//     Term 9 (AT2000-0250)/CC Outputs/Current setpoint value Ch.4 <-> Data Pointer/CurrentSetpointValues[3]
//     Term 9 (AT2000-0250)/CC Outputs/Current setpoint value Ch.5 <-> Data Pointer/CurrentSetpointValues[4]
//     Term 9 (AT2000-0250)/CC Outputs/Current setpoint value Ch.6 <-> Data Pointer/CurrentSetpointValues[5]
//     Term 9 (AT2000-0250)/CC Outputs/Current setpoint value Ch.7 <-> Data Pointer/CurrentSetpointValues[6]
//     Term 9 (AT2000-0250)/CC Outputs/Current setpoint value Ch.8 <-> Data Pointer/CurrentSetpointValues[7]
//     Term 9 (AT2000-0250)/CC Outputs/Current setpoint value Ch.9 <-> Data Pointer/CurrentSetpointValues[8]
//     Term 9 (AT2000-0250)/Term 10 (AT2000-5250)/FB Inputs/Value Channel 01 <-> Data Pointer/RawPositionValues[0]
//     Term 9 (AT2000-0250)/Term 10 (AT2000-5250)/FB Inputs/Value Channel 02 <-> Data Pointer/RawPositionValues[1]
//     Term 9 (AT2000-0250)/Term 10 (AT2000-5250)/FB Inputs/Value Channel 03 <-> Data Pointer/RawPositionValues[2]
//     Term 9 (AT2000-0250)/Term 10 (AT2000-5250)/FB Inputs/Value Channel 04 <-> Data Pointer/RawPositionValues[3]
//     Term 9 (AT2000-0250)/Term 10 (AT2000-5250)/FB Inputs/Value Channel 05 <-> Data Pointer/RawPositionValues[4]
//     Term 9 (AT2000-0250)/Term 10 (AT2000-5250)/FB Inputs/Value Channel 06 <-> Data Pointer/RawPositionValues[5]
//     Term 9 (AT2000-0250)/Term 10 (AT2000-5250)/FB Inputs/Value Channel 07 <-> Data Pointer/RawPositionValues[6]
//     Term 9 (AT2000-0250)/Term 10 (AT2000-5250)/FB Inputs/Value Channel 08 <-> Data Pointer/RawPositionValues[7]
//     Term 9 (AT2000-0250)/Term 10 (AT2000-5250)/FB Inputs/Value Channel 09 <-> Data Pointer/RawPositionValues[8]
//     Term 9 (AT2000-0250)/Term 10 (AT2000-5250)/FB Inputs/Value Channel 10 <-> Data Pointer/RawPositionValues[9]
//     Term 9 (AT2000-0250)/Term 10 (AT2000-5250)/FB Inputs/Value Channel 11 <-> Data Pointer/RawPositionValues[10]
//     Term 9 (AT2000-0250)/Term 10 (AT2000-5250)/FB Inputs/Value Channel 12 <-> Data Pointer/RawPositionValues[11]
//     Term 9 (AT2000-0250)/Term 10 (AT2000-5250)/FB Inputs/Value Channel 13 <-> Data Pointer/RawPositionValues[12]
//     Term 9 (AT2000-0250)/Term 10 (AT2000-5250)/FB Inputs/Value Channel 14 <-> Data Pointer/RawPositionValues[13]
//     Term 9 (AT2000-0250)/Term 10 (AT2000-5250)/FB Inputs/Value Channel 15 <-> Data Pointer/RawPositionValues[14]
//     Term 9 (AT2000-0250)/Term 10 (AT2000-5250)/FB Inputs/Value Channel 16 <-> Data Pointer/RawPositionValues[15]
//     Term 9 (AT2000-0250)/Term 10 (AT2000-5250)/FB Inputs/Value Channel 17 <-> Data Pointer/RawPositionValues[16]
//     Term 9 (AT2000-0250)/Term 10 (AT2000-5250)/FB Inputs/Value Channel 18 <-> Data Pointer/RawPositionValues[17]
//     Term 9 (AT2000-0250)/Term 10 (AT2000-5250)/FB Inputs/Value Channel 19 <-> Data Pointer/RawPositionValues[18]
//     Term 9 (AT2000-0250)/Term 10 (AT2000-5250)/FB Inputs/Value Channel 20 <-> Data Pointer/RawPositionValues[19]
//     Term 9 (AT2000-0250)/Term 10 (AT2000-5250)/FB Inputs/Value Channel 21 <-> Data Pointer/RawPositionValues[20]
//     Term 9 (AT2000-0250)/Term 10 (AT2000-5250)/FB Inputs/Value Channel 22 <-> Data Pointer/RawPositionValues[21]
//     Term 9 (AT2000-0250)/Term 10 (AT2000-5250)/FB Inputs/Value Channel 23 <-> Data Pointer/RawPositionValues[22]
//     Term 9 (AT2000-0250)/Term 10 (AT2000-5250)/FB Inputs/Value Channel 24 <-> Data Pointer/RawPositionValues[23]
//     Term 9 (AT2000-0250)/Term 10 (AT2000-5250)/FB Inputs/Value Channel 25 <-> Data Pointer/RawPositionValues[24]
//     Term 9 (AT2000-0250)/Term 10 (AT2000-5250)/FB Inputs/Value Channel 26 <-> Data Pointer/RawPositionValues[25]
//     Term 9 (AT2000-0250)/Term 10 (AT2000-5250)/FB Inputs/Value Channel 27 <-> Data Pointer/RawPositionValues[26]
//     Term 9 (AT2000-0250)/Term 10 (AT2000-5250)/FB Inputs/Value Channel 28 <-> Data Pointer/RawPositionValues[27]
//     Term 9 (AT2000-0250)/Term 10 (AT2000-5250)/FB Inputs/Value Channel 29 <-> Data Pointer/RawPositionValues[28]
//     Term 9 (AT2000-0250)/Term 10 (AT2000-5250)/FB Inputs/Value Channel 30 <-> Data Pointer/RawPositionValues[29]
//     Term 9 (AT2000-0250)/Term 10 (AT2000-5250)/FB Inputs/Value Channel 31 <-> Data Pointer/RawPositionValues[30]
//     Term 9 (AT2000-0250)/Term 10 (AT2000-5250)/FB Inputs/Value Channel 32 <-> Data Pointer/RawPositionValues[31]
//   (this object) <-> TcCOM Objects/XtsProcessingUnit 1/Part 1/Module 6
//     Term 11 (AT2000-0250)/CC Inputs/Current actual value Ch.1 <-> Data Pointer/CurrentActualValues[0]
//     Term 11 (AT2000-0250)/CC Inputs/Current actual value Ch.10 <-> Data Pointer/CurrentActualValues[9]
//     Term 11 (AT2000-0250)/CC Inputs/Current actual value Ch.11 <-> Data Pointer/CurrentActualValues[10]
//     Term 11 (AT2000-0250)/CC Inputs/Current actual value Ch.12 <-> Data Pointer/CurrentActualValues[11]
//     Term 11 (AT2000-0250)/CC Inputs/Current actual value Ch.13 <-> Data Pointer/CurrentActualValues[12]
//     Term 11 (AT2000-0250)/CC Inputs/Current actual value Ch.14 <-> Data Pointer/CurrentActualValues[13]
//     Term 11 (AT2000-0250)/CC Inputs/Current actual value Ch.15 <-> Data Pointer/CurrentActualValues[14]
//     Term 11 (AT2000-0250)/CC Inputs/Current actual value Ch.2 <-> Data Pointer/CurrentActualValues[1]
//     Term 11 (AT2000-0250)/CC Inputs/Current actual value Ch.3 <-> Data Pointer/CurrentActualValues[2]
//     Term 11 (AT2000-0250)/CC Inputs/Current actual value Ch.4 <-> Data Pointer/CurrentActualValues[3]
//     Term 11 (AT2000-0250)/CC Inputs/Current actual value Ch.5 <-> Data Pointer/CurrentActualValues[4]
//     Term 11 (AT2000-0250)/CC Inputs/Current actual value Ch.6 <-> Data Pointer/CurrentActualValues[5]
//     Term 11 (AT2000-0250)/CC Inputs/Current actual value Ch.7 <-> Data Pointer/CurrentActualValues[6]
//     Term 11 (AT2000-0250)/CC Inputs/Current actual value Ch.8 <-> Data Pointer/CurrentActualValues[7]
//     Term 11 (AT2000-0250)/CC Inputs/Current actual value Ch.9 <-> Data Pointer/CurrentActualValues[8]
//     Term 11 (AT2000-0250)/CC Inputs/Status <-> Data Pointer/Status
//     Term 11 (AT2000-0250)/CC Outputs/Control <-> Data Pointer/Control
//     Term 11 (AT2000-0250)/CC Outputs/Current setpoint value Ch.1 <-> Data Pointer/CurrentSetpointValues[0]
//     Term 11 (AT2000-0250)/CC Outputs/Current setpoint value Ch.10 <-> Data Pointer/CurrentSetpointValues[9]
//     Term 11 (AT2000-0250)/CC Outputs/Current setpoint value Ch.11 <-> Data Pointer/CurrentSetpointValues[10]
//     Term 11 (AT2000-0250)/CC Outputs/Current setpoint value Ch.12 <-> Data Pointer/CurrentSetpointValues[11]
//     Term 11 (AT2000-0250)/CC Outputs/Current setpoint value Ch.13 <-> Data Pointer/CurrentSetpointValues[12]
//     Term 11 (AT2000-0250)/CC Outputs/Current setpoint value Ch.14 <-> Data Pointer/CurrentSetpointValues[13]
//     Term 11 (AT2000-0250)/CC Outputs/Current setpoint value Ch.15 <-> Data Pointer/CurrentSetpointValues[14]
//     Term 11 (AT2000-0250)/CC Outputs/Current setpoint value Ch.2 <-> Data Pointer/CurrentSetpointValues[1]
//     Term 11 (AT2000-0250)/CC Outputs/Current setpoint value Ch.3 <-> Data Pointer/CurrentSetpointValues[2]
//     Term 11 (AT2000-0250)/CC Outputs/Current setpoint value Ch.4 <-> Data Pointer/CurrentSetpointValues[3]
//     Term 11 (AT2000-0250)/CC Outputs/Current setpoint value Ch.5 <-> Data Pointer/CurrentSetpointValues[4]
//     Term 11 (AT2000-0250)/CC Outputs/Current setpoint value Ch.6 <-> Data Pointer/CurrentSetpointValues[5]
//     Term 11 (AT2000-0250)/CC Outputs/Current setpoint value Ch.7 <-> Data Pointer/CurrentSetpointValues[6]
//     Term 11 (AT2000-0250)/CC Outputs/Current setpoint value Ch.8 <-> Data Pointer/CurrentSetpointValues[7]
//     Term 11 (AT2000-0250)/CC Outputs/Current setpoint value Ch.9 <-> Data Pointer/CurrentSetpointValues[8]
//     Term 11 (AT2000-0250)/Term 12 (AT2000-5250)/FB Inputs/Value Channel 01 <-> Data Pointer/RawPositionValues[0]
//     Term 11 (AT2000-0250)/Term 12 (AT2000-5250)/FB Inputs/Value Channel 02 <-> Data Pointer/RawPositionValues[1]
//     Term 11 (AT2000-0250)/Term 12 (AT2000-5250)/FB Inputs/Value Channel 03 <-> Data Pointer/RawPositionValues[2]
//     Term 11 (AT2000-0250)/Term 12 (AT2000-5250)/FB Inputs/Value Channel 04 <-> Data Pointer/RawPositionValues[3]
//     Term 11 (AT2000-0250)/Term 12 (AT2000-5250)/FB Inputs/Value Channel 05 <-> Data Pointer/RawPositionValues[4]
//     Term 11 (AT2000-0250)/Term 12 (AT2000-5250)/FB Inputs/Value Channel 06 <-> Data Pointer/RawPositionValues[5]
//     Term 11 (AT2000-0250)/Term 12 (AT2000-5250)/FB Inputs/Value Channel 07 <-> Data Pointer/RawPositionValues[6]
//     Term 11 (AT2000-0250)/Term 12 (AT2000-5250)/FB Inputs/Value Channel 08 <-> Data Pointer/RawPositionValues[7]
//     Term 11 (AT2000-0250)/Term 12 (AT2000-5250)/FB Inputs/Value Channel 09 <-> Data Pointer/RawPositionValues[8]
//     Term 11 (AT2000-0250)/Term 12 (AT2000-5250)/FB Inputs/Value Channel 10 <-> Data Pointer/RawPositionValues[9]
//     Term 11 (AT2000-0250)/Term 12 (AT2000-5250)/FB Inputs/Value Channel 11 <-> Data Pointer/RawPositionValues[10]
//     Term 11 (AT2000-0250)/Term 12 (AT2000-5250)/FB Inputs/Value Channel 12 <-> Data Pointer/RawPositionValues[11]
//     Term 11 (AT2000-0250)/Term 12 (AT2000-5250)/FB Inputs/Value Channel 13 <-> Data Pointer/RawPositionValues[12]
//     Term 11 (AT2000-0250)/Term 12 (AT2000-5250)/FB Inputs/Value Channel 14 <-> Data Pointer/RawPositionValues[13]
//     Term 11 (AT2000-0250)/Term 12 (AT2000-5250)/FB Inputs/Value Channel 15 <-> Data Pointer/RawPositionValues[14]
//     Term 11 (AT2000-0250)/Term 12 (AT2000-5250)/FB Inputs/Value Channel 16 <-> Data Pointer/RawPositionValues[15]
//     Term 11 (AT2000-0250)/Term 12 (AT2000-5250)/FB Inputs/Value Channel 17 <-> Data Pointer/RawPositionValues[16]
//     Term 11 (AT2000-0250)/Term 12 (AT2000-5250)/FB Inputs/Value Channel 18 <-> Data Pointer/RawPositionValues[17]
//     Term 11 (AT2000-0250)/Term 12 (AT2000-5250)/FB Inputs/Value Channel 19 <-> Data Pointer/RawPositionValues[18]
//     Term 11 (AT2000-0250)/Term 12 (AT2000-5250)/FB Inputs/Value Channel 20 <-> Data Pointer/RawPositionValues[19]
//     Term 11 (AT2000-0250)/Term 12 (AT2000-5250)/FB Inputs/Value Channel 21 <-> Data Pointer/RawPositionValues[20]
//     Term 11 (AT2000-0250)/Term 12 (AT2000-5250)/FB Inputs/Value Channel 22 <-> Data Pointer/RawPositionValues[21]
//     Term 11 (AT2000-0250)/Term 12 (AT2000-5250)/FB Inputs/Value Channel 23 <-> Data Pointer/RawPositionValues[22]
//     Term 11 (AT2000-0250)/Term 12 (AT2000-5250)/FB Inputs/Value Channel 24 <-> Data Pointer/RawPositionValues[23]
//     Term 11 (AT2000-0250)/Term 12 (AT2000-5250)/FB Inputs/Value Channel 25 <-> Data Pointer/RawPositionValues[24]
//     Term 11 (AT2000-0250)/Term 12 (AT2000-5250)/FB Inputs/Value Channel 26 <-> Data Pointer/RawPositionValues[25]
//     Term 11 (AT2000-0250)/Term 12 (AT2000-5250)/FB Inputs/Value Channel 27 <-> Data Pointer/RawPositionValues[26]
//     Term 11 (AT2000-0250)/Term 12 (AT2000-5250)/FB Inputs/Value Channel 28 <-> Data Pointer/RawPositionValues[27]
//     Term 11 (AT2000-0250)/Term 12 (AT2000-5250)/FB Inputs/Value Channel 29 <-> Data Pointer/RawPositionValues[28]
//     Term 11 (AT2000-0250)/Term 12 (AT2000-5250)/FB Inputs/Value Channel 30 <-> Data Pointer/RawPositionValues[29]
//     Term 11 (AT2000-0250)/Term 12 (AT2000-5250)/FB Inputs/Value Channel 31 <-> Data Pointer/RawPositionValues[30]
//     Term 11 (AT2000-0250)/Term 12 (AT2000-5250)/FB Inputs/Value Channel 32 <-> Data Pointer/RawPositionValues[31]
//   (this object) <-> TcCOM Objects/XtsProcessingUnit 1/Part 1/Module 7
//     Term 13 (AT2050-0500)/CC Inputs/Current actual value Ch.1 <-> Data Pointer/CurrentActualValues[0]
//     Term 13 (AT2050-0500)/CC Inputs/Current actual value Ch.10 <-> Data Pointer/CurrentActualValues[9]
//     Term 13 (AT2050-0500)/CC Inputs/Current actual value Ch.11 <-> Data Pointer/CurrentActualValues[10]
//     Term 13 (AT2050-0500)/CC Inputs/Current actual value Ch.12 <-> Data Pointer/CurrentActualValues[11]
//     Term 13 (AT2050-0500)/CC Inputs/Current actual value Ch.13 <-> Data Pointer/CurrentActualValues[12]
//     Term 13 (AT2050-0500)/CC Inputs/Current actual value Ch.14 <-> Data Pointer/CurrentActualValues[13]
//     Term 13 (AT2050-0500)/CC Inputs/Current actual value Ch.15 <-> Data Pointer/CurrentActualValues[14]
//     Term 13 (AT2050-0500)/CC Inputs/Current actual value Ch.2 <-> Data Pointer/CurrentActualValues[1]
//     Term 13 (AT2050-0500)/CC Inputs/Current actual value Ch.3 <-> Data Pointer/CurrentActualValues[2]
//     Term 13 (AT2050-0500)/CC Inputs/Current actual value Ch.4 <-> Data Pointer/CurrentActualValues[3]
//     Term 13 (AT2050-0500)/CC Inputs/Current actual value Ch.5 <-> Data Pointer/CurrentActualValues[4]
//     Term 13 (AT2050-0500)/CC Inputs/Current actual value Ch.6 <-> Data Pointer/CurrentActualValues[5]
//     Term 13 (AT2050-0500)/CC Inputs/Current actual value Ch.7 <-> Data Pointer/CurrentActualValues[6]
//     Term 13 (AT2050-0500)/CC Inputs/Current actual value Ch.8 <-> Data Pointer/CurrentActualValues[7]
//     Term 13 (AT2050-0500)/CC Inputs/Current actual value Ch.9 <-> Data Pointer/CurrentActualValues[8]
//     Term 13 (AT2050-0500)/CC Inputs/Status <-> Data Pointer/Status
//     Term 13 (AT2050-0500)/CC Outputs/Control <-> Data Pointer/Control
//     Term 13 (AT2050-0500)/CC Outputs/Current setpoint value Ch.1 <-> Data Pointer/CurrentSetpointValues[0]
//     Term 13 (AT2050-0500)/CC Outputs/Current setpoint value Ch.10 <-> Data Pointer/CurrentSetpointValues[9]
//     Term 13 (AT2050-0500)/CC Outputs/Current setpoint value Ch.11 <-> Data Pointer/CurrentSetpointValues[10]
//     Term 13 (AT2050-0500)/CC Outputs/Current setpoint value Ch.12 <-> Data Pointer/CurrentSetpointValues[11]
//     Term 13 (AT2050-0500)/CC Outputs/Current setpoint value Ch.13 <-> Data Pointer/CurrentSetpointValues[12]
//     Term 13 (AT2050-0500)/CC Outputs/Current setpoint value Ch.14 <-> Data Pointer/CurrentSetpointValues[13]
//     Term 13 (AT2050-0500)/CC Outputs/Current setpoint value Ch.15 <-> Data Pointer/CurrentSetpointValues[14]
//     Term 13 (AT2050-0500)/CC Outputs/Current setpoint value Ch.2 <-> Data Pointer/CurrentSetpointValues[1]
//     Term 13 (AT2050-0500)/CC Outputs/Current setpoint value Ch.3 <-> Data Pointer/CurrentSetpointValues[2]
//     Term 13 (AT2050-0500)/CC Outputs/Current setpoint value Ch.4 <-> Data Pointer/CurrentSetpointValues[3]
//     Term 13 (AT2050-0500)/CC Outputs/Current setpoint value Ch.5 <-> Data Pointer/CurrentSetpointValues[4]
//     Term 13 (AT2050-0500)/CC Outputs/Current setpoint value Ch.6 <-> Data Pointer/CurrentSetpointValues[5]
//     Term 13 (AT2050-0500)/CC Outputs/Current setpoint value Ch.7 <-> Data Pointer/CurrentSetpointValues[6]
//     Term 13 (AT2050-0500)/CC Outputs/Current setpoint value Ch.8 <-> Data Pointer/CurrentSetpointValues[7]
//     Term 13 (AT2050-0500)/CC Outputs/Current setpoint value Ch.9 <-> Data Pointer/CurrentSetpointValues[8]
//     Term 13 (AT2050-0500)/Term 14 (AT2050-5500)/FB Inputs/Value Channel 01 <-> Data Pointer/RawPositionValues[0]
//     Term 13 (AT2050-0500)/Term 14 (AT2050-5500)/FB Inputs/Value Channel 02 <-> Data Pointer/RawPositionValues[1]
//     Term 13 (AT2050-0500)/Term 14 (AT2050-5500)/FB Inputs/Value Channel 03 <-> Data Pointer/RawPositionValues[2]
//     Term 13 (AT2050-0500)/Term 14 (AT2050-5500)/FB Inputs/Value Channel 04 <-> Data Pointer/RawPositionValues[3]
//     Term 13 (AT2050-0500)/Term 14 (AT2050-5500)/FB Inputs/Value Channel 05 <-> Data Pointer/RawPositionValues[4]
//     Term 13 (AT2050-0500)/Term 14 (AT2050-5500)/FB Inputs/Value Channel 06 <-> Data Pointer/RawPositionValues[5]
//     Term 13 (AT2050-0500)/Term 14 (AT2050-5500)/FB Inputs/Value Channel 07 <-> Data Pointer/RawPositionValues[6]
//     Term 13 (AT2050-0500)/Term 14 (AT2050-5500)/FB Inputs/Value Channel 08 <-> Data Pointer/RawPositionValues[7]
//     Term 13 (AT2050-0500)/Term 14 (AT2050-5500)/FB Inputs/Value Channel 09 <-> Data Pointer/RawPositionValues[8]
//     Term 13 (AT2050-0500)/Term 14 (AT2050-5500)/FB Inputs/Value Channel 10 <-> Data Pointer/RawPositionValues[9]
//     Term 13 (AT2050-0500)/Term 14 (AT2050-5500)/FB Inputs/Value Channel 11 <-> Data Pointer/RawPositionValues[10]
//     Term 13 (AT2050-0500)/Term 14 (AT2050-5500)/FB Inputs/Value Channel 12 <-> Data Pointer/RawPositionValues[11]
//     Term 13 (AT2050-0500)/Term 14 (AT2050-5500)/FB Inputs/Value Channel 13 <-> Data Pointer/RawPositionValues[12]
//     Term 13 (AT2050-0500)/Term 14 (AT2050-5500)/FB Inputs/Value Channel 14 <-> Data Pointer/RawPositionValues[13]
//     Term 13 (AT2050-0500)/Term 14 (AT2050-5500)/FB Inputs/Value Channel 15 <-> Data Pointer/RawPositionValues[14]
//     Term 13 (AT2050-0500)/Term 14 (AT2050-5500)/FB Inputs/Value Channel 16 <-> Data Pointer/RawPositionValues[15]
//     Term 13 (AT2050-0500)/Term 14 (AT2050-5500)/FB Inputs/Value Channel 17 <-> Data Pointer/RawPositionValues[16]
//     Term 13 (AT2050-0500)/Term 14 (AT2050-5500)/FB Inputs/Value Channel 18 <-> Data Pointer/RawPositionValues[17]
//     Term 13 (AT2050-0500)/Term 14 (AT2050-5500)/FB Inputs/Value Channel 19 <-> Data Pointer/RawPositionValues[18]
//     Term 13 (AT2050-0500)/Term 14 (AT2050-5500)/FB Inputs/Value Channel 20 <-> Data Pointer/RawPositionValues[19]
//     Term 13 (AT2050-0500)/Term 14 (AT2050-5500)/FB Inputs/Value Channel 21 <-> Data Pointer/RawPositionValues[20]
//     Term 13 (AT2050-0500)/Term 14 (AT2050-5500)/FB Inputs/Value Channel 22 <-> Data Pointer/RawPositionValues[21]
//     Term 13 (AT2050-0500)/Term 14 (AT2050-5500)/FB Inputs/Value Channel 23 <-> Data Pointer/RawPositionValues[22]
//     Term 13 (AT2050-0500)/Term 14 (AT2050-5500)/FB Inputs/Value Channel 24 <-> Data Pointer/RawPositionValues[23]
//     Term 13 (AT2050-0500)/Term 14 (AT2050-5500)/FB Inputs/Value Channel 25 <-> Data Pointer/RawPositionValues[24]
//     Term 13 (AT2050-0500)/Term 14 (AT2050-5500)/FB Inputs/Value Channel 26 <-> Data Pointer/RawPositionValues[25]
//     Term 13 (AT2050-0500)/Term 14 (AT2050-5500)/FB Inputs/Value Channel 27 <-> Data Pointer/RawPositionValues[26]
//     Term 13 (AT2050-0500)/Term 14 (AT2050-5500)/FB Inputs/Value Channel 28 <-> Data Pointer/RawPositionValues[27]
//     Term 13 (AT2050-0500)/Term 14 (AT2050-5500)/FB Inputs/Value Channel 29 <-> Data Pointer/RawPositionValues[28]
//     Term 13 (AT2050-0500)/Term 14 (AT2050-5500)/FB Inputs/Value Channel 30 <-> Data Pointer/RawPositionValues[29]
//     Term 13 (AT2050-0500)/Term 14 (AT2050-5500)/FB Inputs/Value Channel 31 <-> Data Pointer/RawPositionValues[30]
//     Term 13 (AT2050-0500)/Term 14 (AT2050-5500)/FB Inputs/Value Channel 32 <-> Data Pointer/RawPositionValues[31]
//   (this object) <-> TcCOM Objects/XtsProcessingUnit 1/Part 1/Module 8
//     Term 15 (AT2050-0501)/CC Inputs/Current actual value Ch.1 <-> Data Pointer/CurrentActualValues[0]
//     Term 15 (AT2050-0501)/CC Inputs/Current actual value Ch.10 <-> Data Pointer/CurrentActualValues[9]
//     Term 15 (AT2050-0501)/CC Inputs/Current actual value Ch.11 <-> Data Pointer/CurrentActualValues[10]
//     Term 15 (AT2050-0501)/CC Inputs/Current actual value Ch.12 <-> Data Pointer/CurrentActualValues[11]
//     Term 15 (AT2050-0501)/CC Inputs/Current actual value Ch.13 <-> Data Pointer/CurrentActualValues[12]
//     Term 15 (AT2050-0501)/CC Inputs/Current actual value Ch.14 <-> Data Pointer/CurrentActualValues[13]
//     Term 15 (AT2050-0501)/CC Inputs/Current actual value Ch.15 <-> Data Pointer/CurrentActualValues[14]
//     Term 15 (AT2050-0501)/CC Inputs/Current actual value Ch.2 <-> Data Pointer/CurrentActualValues[1]
//     Term 15 (AT2050-0501)/CC Inputs/Current actual value Ch.3 <-> Data Pointer/CurrentActualValues[2]
//     Term 15 (AT2050-0501)/CC Inputs/Current actual value Ch.4 <-> Data Pointer/CurrentActualValues[3]
//     Term 15 (AT2050-0501)/CC Inputs/Current actual value Ch.5 <-> Data Pointer/CurrentActualValues[4]
//     Term 15 (AT2050-0501)/CC Inputs/Current actual value Ch.6 <-> Data Pointer/CurrentActualValues[5]
//     Term 15 (AT2050-0501)/CC Inputs/Current actual value Ch.7 <-> Data Pointer/CurrentActualValues[6]
//     Term 15 (AT2050-0501)/CC Inputs/Current actual value Ch.8 <-> Data Pointer/CurrentActualValues[7]
//     Term 15 (AT2050-0501)/CC Inputs/Current actual value Ch.9 <-> Data Pointer/CurrentActualValues[8]
//     Term 15 (AT2050-0501)/CC Inputs/Status <-> Data Pointer/Status
//     Term 15 (AT2050-0501)/CC Outputs/Control <-> Data Pointer/Control
//     Term 15 (AT2050-0501)/CC Outputs/Current setpoint value Ch.1 <-> Data Pointer/CurrentSetpointValues[0]
//     Term 15 (AT2050-0501)/CC Outputs/Current setpoint value Ch.10 <-> Data Pointer/CurrentSetpointValues[9]
//     Term 15 (AT2050-0501)/CC Outputs/Current setpoint value Ch.11 <-> Data Pointer/CurrentSetpointValues[10]
//     Term 15 (AT2050-0501)/CC Outputs/Current setpoint value Ch.12 <-> Data Pointer/CurrentSetpointValues[11]
//     Term 15 (AT2050-0501)/CC Outputs/Current setpoint value Ch.13 <-> Data Pointer/CurrentSetpointValues[12]
//     Term 15 (AT2050-0501)/CC Outputs/Current setpoint value Ch.14 <-> Data Pointer/CurrentSetpointValues[13]
//     Term 15 (AT2050-0501)/CC Outputs/Current setpoint value Ch.15 <-> Data Pointer/CurrentSetpointValues[14]
//     Term 15 (AT2050-0501)/CC Outputs/Current setpoint value Ch.2 <-> Data Pointer/CurrentSetpointValues[1]
//     Term 15 (AT2050-0501)/CC Outputs/Current setpoint value Ch.3 <-> Data Pointer/CurrentSetpointValues[2]
//     Term 15 (AT2050-0501)/CC Outputs/Current setpoint value Ch.4 <-> Data Pointer/CurrentSetpointValues[3]
//     Term 15 (AT2050-0501)/CC Outputs/Current setpoint value Ch.5 <-> Data Pointer/CurrentSetpointValues[4]
//     Term 15 (AT2050-0501)/CC Outputs/Current setpoint value Ch.6 <-> Data Pointer/CurrentSetpointValues[5]
//     Term 15 (AT2050-0501)/CC Outputs/Current setpoint value Ch.7 <-> Data Pointer/CurrentSetpointValues[6]
//     Term 15 (AT2050-0501)/CC Outputs/Current setpoint value Ch.8 <-> Data Pointer/CurrentSetpointValues[7]
//     Term 15 (AT2050-0501)/CC Outputs/Current setpoint value Ch.9 <-> Data Pointer/CurrentSetpointValues[8]
//     Term 15 (AT2050-0501)/Term 16 (AT2050-5501)/FB Inputs/Value Channel 01 <-> Data Pointer/RawPositionValues[0]
//     Term 15 (AT2050-0501)/Term 16 (AT2050-5501)/FB Inputs/Value Channel 02 <-> Data Pointer/RawPositionValues[1]
//     Term 15 (AT2050-0501)/Term 16 (AT2050-5501)/FB Inputs/Value Channel 03 <-> Data Pointer/RawPositionValues[2]
//     Term 15 (AT2050-0501)/Term 16 (AT2050-5501)/FB Inputs/Value Channel 04 <-> Data Pointer/RawPositionValues[3]
//     Term 15 (AT2050-0501)/Term 16 (AT2050-5501)/FB Inputs/Value Channel 05 <-> Data Pointer/RawPositionValues[4]
//     Term 15 (AT2050-0501)/Term 16 (AT2050-5501)/FB Inputs/Value Channel 06 <-> Data Pointer/RawPositionValues[5]
//     Term 15 (AT2050-0501)/Term 16 (AT2050-5501)/FB Inputs/Value Channel 07 <-> Data Pointer/RawPositionValues[6]
//     Term 15 (AT2050-0501)/Term 16 (AT2050-5501)/FB Inputs/Value Channel 08 <-> Data Pointer/RawPositionValues[7]
//     Term 15 (AT2050-0501)/Term 16 (AT2050-5501)/FB Inputs/Value Channel 09 <-> Data Pointer/RawPositionValues[8]
//     Term 15 (AT2050-0501)/Term 16 (AT2050-5501)/FB Inputs/Value Channel 10 <-> Data Pointer/RawPositionValues[9]
//     Term 15 (AT2050-0501)/Term 16 (AT2050-5501)/FB Inputs/Value Channel 11 <-> Data Pointer/RawPositionValues[10]
//     Term 15 (AT2050-0501)/Term 16 (AT2050-5501)/FB Inputs/Value Channel 12 <-> Data Pointer/RawPositionValues[11]
//     Term 15 (AT2050-0501)/Term 16 (AT2050-5501)/FB Inputs/Value Channel 13 <-> Data Pointer/RawPositionValues[12]
//     Term 15 (AT2050-0501)/Term 16 (AT2050-5501)/FB Inputs/Value Channel 14 <-> Data Pointer/RawPositionValues[13]
//     Term 15 (AT2050-0501)/Term 16 (AT2050-5501)/FB Inputs/Value Channel 15 <-> Data Pointer/RawPositionValues[14]
//     Term 15 (AT2050-0501)/Term 16 (AT2050-5501)/FB Inputs/Value Channel 16 <-> Data Pointer/RawPositionValues[15]
//     Term 15 (AT2050-0501)/Term 16 (AT2050-5501)/FB Inputs/Value Channel 17 <-> Data Pointer/RawPositionValues[16]
//     Term 15 (AT2050-0501)/Term 16 (AT2050-5501)/FB Inputs/Value Channel 18 <-> Data Pointer/RawPositionValues[17]
//     Term 15 (AT2050-0501)/Term 16 (AT2050-5501)/FB Inputs/Value Channel 19 <-> Data Pointer/RawPositionValues[18]
//     Term 15 (AT2050-0501)/Term 16 (AT2050-5501)/FB Inputs/Value Channel 20 <-> Data Pointer/RawPositionValues[19]
//     Term 15 (AT2050-0501)/Term 16 (AT2050-5501)/FB Inputs/Value Channel 21 <-> Data Pointer/RawPositionValues[20]
//     Term 15 (AT2050-0501)/Term 16 (AT2050-5501)/FB Inputs/Value Channel 22 <-> Data Pointer/RawPositionValues[21]
//     Term 15 (AT2050-0501)/Term 16 (AT2050-5501)/FB Inputs/Value Channel 23 <-> Data Pointer/RawPositionValues[22]
//     Term 15 (AT2050-0501)/Term 16 (AT2050-5501)/FB Inputs/Value Channel 24 <-> Data Pointer/RawPositionValues[23]
//     Term 15 (AT2050-0501)/Term 16 (AT2050-5501)/FB Inputs/Value Channel 25 <-> Data Pointer/RawPositionValues[24]
//     Term 15 (AT2050-0501)/Term 16 (AT2050-5501)/FB Inputs/Value Channel 26 <-> Data Pointer/RawPositionValues[25]
//     Term 15 (AT2050-0501)/Term 16 (AT2050-5501)/FB Inputs/Value Channel 27 <-> Data Pointer/RawPositionValues[26]
//     Term 15 (AT2050-0501)/Term 16 (AT2050-5501)/FB Inputs/Value Channel 28 <-> Data Pointer/RawPositionValues[27]
//     Term 15 (AT2050-0501)/Term 16 (AT2050-5501)/FB Inputs/Value Channel 29 <-> Data Pointer/RawPositionValues[28]
//     Term 15 (AT2050-0501)/Term 16 (AT2050-5501)/FB Inputs/Value Channel 30 <-> Data Pointer/RawPositionValues[29]
//     Term 15 (AT2050-0501)/Term 16 (AT2050-5501)/FB Inputs/Value Channel 31 <-> Data Pointer/RawPositionValues[30]
//     Term 15 (AT2050-0501)/Term 16 (AT2050-5501)/FB Inputs/Value Channel 32 <-> Data Pointer/RawPositionValues[31]

// ---- GVLs/Param.TcGVL
{attribute 'qualified_only'}
VAR_GLOBAL CONSTANT
	// The following should be set to a value **equal to or greater than** the number of objects needed
	MAX_MOVERS   			: USINT := 100;	// Movers
	MAX_POSITIONTRIGGERS	: USINT := 100;	// Position triggers
	MAX_STATIONS			: USINT := 100;	// Stations
	MAX_ZONES				: USINT := 100;	// Zones
	
	// The following should be set to a value **equal to or greater than** the number of objectives needed
	// it's also possible to declare additional stations, zones and position triggers in MAIN
	NUM_MOVERLISTS			: USINT := 10;	// Mover Lists
	NUM_POSITIONTRIGGERS	: USINT := 10;	// Position Triggers
	NUM_STATIONS			: USINT := 10;	// Stations
	NUM_ZONES				: USINT := 10;	// Zones
	
	NUM_TRACKS				: USINT	:= 1;	// Tracks (Typically 1)
	DEFAULT_TRACK			: USINT := 1;	// Default track for movers, stations, zones and position triggers

	PART_ARRAY_SIZE			: UDINT := 100;
	AUTO_POPULATE_STATIONS  : BOOL := TRUE; // use the Station[x] array to label stations on the visualization. Turn off if manually entering stations in the configurator.
	
	// statistics weighted average
	ALPHA_EMA				: LREAL := 0.1;
END_VAR

// ---- POUs/MAIN.TcPOU

      PROGRAM MAIN
VAR	
	// declare XTS with <number of movers>
	XTS				: FB_XTS<6>;
	// Machine
	State			: MachineState_enum;

	// ========= Example Application Variables =========

    nextStation 			: USINT := 4;
                    	
	StationTimer 			: ARRAY[0..Param.NUM_STATIONS] OF TON; // timer blocks, for station dwells
	RecoveryComplete		: BOOL;
	
	Trig0MoverIndex			: UDINT;
	Trig0MoverPosLag		: LREAL;
END_VAR


        
(* ======================================================================================

--- XTS Starter Project ---

This MAIN (PRG) is intended to serve as an example, which can be modified to suit your specific application.

No programming changes should be necessary inside the provided XTS objects / function block definitions.
They are intended to be simply instantiated and controlled via the provided methods and properties.
However the objects are provided as open-source for modification and extension as needed.

Documentation for these objects can be found online at:
https://beckhoff-usa-community.github.io/XTS_Base/

Bug reports, new feature requests, and general feedback is always welcome on our Github page.
For any other questions, please reach out to your local Application Engineer.

Version 2.1.0 of XTS_Base has been tested with:

- TwinCAT XAE v4026.20.1
- TF5850 XTS v4.4.5
- TF5410 Advanced Motion v3.4.19

- XTS Application Group | Beckhoff USA

====================================================================================== *)

(*
All sample code provided by Beckhoff Automation LLC are for illustrative purposes only
and are provided “as is” and without any warranties, express or implied. Actual
implementations in applications will vary significantly. Beckhoff Automation LLC shall
have no liability for, and does not waive any rights in relation to, any code samples that it
provides or the use of such code samples for any purpose.
*)

// main state machine
CASE State OF 

	// off (idle) state, waiting for enable command
	MS_OFF:
		// wait for enable command
		IF MainCommands.Enable AND XTS.System.EnvironmentIsReady THEN
			// initialize stations, positions and triggers
			Initializing();
			// enable the XTS
			XTS.Enable				:= TRUE;
			State					:= MS_RESTARTING;
		END_IF
		
	MS_RESTARTING:
		// restart the system by enabling the XTS and waiting for it to complete
		IF NOT MainCommands.Enable THEN
			// disable triggered, pass to xts and stop the movers
			XTS.Enable				:= FALSE;
			State					:= MS_STOPPED;
		ELSIF XTS.State = XTS_ENABLED THEN
			// enable complete move to enabled
			State		:= MS_ENABLED;
		END_IF


	MS_ENABLED:
		// XTS is enabled, wait for start command
		IF NOT MainCommands.Enable THEN
			XTS.Enable				:= FALSE;
			State					:= MS_STOPPED;
		ELSIF MainCommands.Start THEN
			// reset the recovery complete flag
			RecoveryComplete		:= FALSE;
			// move to next state
			State					:= MS_ONESHOT_RECOVER;
		END_IF
		
	MS_ONESHOT_RECOVER:
		// one time commands before starting typical process motions
		RecoverOneshot();
		State := MS_RECOVERING;
		
	MS_RECOVERING:
		// wait for any recovery actions to complete
		Recovering();
		// test for errors, commands or recovery complete
		IF MainCommands.Stop THEN
			// respond to stop command
			MainCommands.Start		:= FALSE;
			XTS.System.CompleteMoverList.HaltAll();
            State         	:= MS_STOPPED;
        ELSIF NOT MainCommands.Enable THEN
			// respond to loss of enable
            XTS.Enable		:= FALSE;
			XTS.System.CompleteMoverList.HaltAll();
            State          			:= MS_STOPPED;
		ELSIF RecoveryComplete THEN
			// clear any position trigers that were not consumed during recovery
			XTS.System.MuteAllPositionTriggers();
			// recovery sequence is complete, move on to run state
			State					:= MS_RUNNING;
        END_IF

	MS_RUNNING:
		// run the station-to-station mover logic
		StationLogic();
		
		// monitor for disable or stop
		IF NOT MainCommands.Enable THEN
			XTS.Enable				:= FALSE;
			XTS.System.CompleteMoverList.HaltAll();
			State					:= MS_STOPPED;
		ELSIF MainCommands.Stop THEN
			MainCommands.Start		:= FALSE;
			XTS.System.CompleteMoverList.HaltAll();
			State					:= MS_STOPPED;
		END_IF

	MS_STOPPED:
		// movers are stopped, but XTS is still enabled
		// wait for restart, disable or error disable
		IF XTS.State <> XTS_ENABLED AND MainCommands.Enable THEN
			State					:= MS_ERROR;
		ELSIF NOT MainCommands.Enable THEN
			XTS.Enable 				:= FALSE;
		ELSIF  MainCommands.Start THEN
			MainCommands.Stop		:= FALSE;
			State					:= MS_ONESHOT_RECOVER;
		END_IF
		IF XTS.State = XTS_DISABLED THEN
			State					:= MS_OFF;
		END_IF;
		
	MS_ERROR:
		// and error has occured
		// the recovery from this is application dependent and can range from disabling and re-enabling the XTS
		// to specific needs for each mover/station/zone and how to clear them of tooling and/or defective product
		
		// the simplest form of error handling where the XTS is disabled and re-enabled is available as this commented code below
// 		IF NOT MainCommands.Enable THEN
// 			XTS.Enable := FALSE;
// 			State					:= MS_OFF;
// 		END_IF;
			
	
END_CASE

// call the main XTS logic
XTS.CyclicLogic();

ACTION Initializing:

          // XTS Object Init
XTS.Station[0].Position 		:= 5;
XTS.Station[1].Position 		:= 750;
XTS.Station[2].Position 		:= 1200;
XTS.Station[3].Position 		:= 1300;
XTS.Station[4].Position 		:= 1400;

// station names
XTS.Station[0].Description		:= 'Load Top';
XTS.Station[1].Description		:= 'Load Bottom';
XTS.Station[2].Description		:= 'Weld A';
XTS.Station[3].Description		:= 'Weld B';
XTS.Station[4].Description		:= 'Weld C';

// speed changes in corners
XTS.PositionTrigger[0].Position := 1500;
XTS.PositionTrigger[1].Position := 2000;
XTS.PositionTrigger[2].Position := 3500;

// recover trigger near station 0
XTS.PositionTrigger[3].Position := XTS.Station[0].Position + 2.0;

// window around station 0 for startup
XTS.Zone[0].StartPosition		:= XTS.Station[0].Position - 1.0;
XTS.Zone[0].EndPosition   		:= XTS.Station[0].Position + 1.0;

XTS.InitialParameterSet.Velocity		:= 1000;		// mm/s
XTS.InitialParameterSet.Acceleration	:= 10_000;		// mm/s2
XTS.InitialParameterSet.Deceleration	:= 10_000;		// mm/s2
XTS.InitialParameterSet.Jerk			:= 100_000;		// mm/s3
XTS.InitialParameterSet.Gap				:= 85;			// mm
XTS.InitialParameterSet.Direction		:= Tc3_Mc3Definitions.MC_Direction.mcDirectionPositive;

MainCommands.lowVelocity	:= 300;
MainCommands.mediumVelocity	:= 800;
MainCommands.highVelocity	:= 1200;
END_ACTION

ACTION Recovering:

          // this state is called until all movers have completed their desired recovery tasks

// wait for all movers to reach the standstill state and one mover at station 0
IF (XTS.System.CompleteMoverList.IsAllMoversHalted AND XTS.Station[0].MoverInPosition) THEN
	RecoveryComplete := TRUE;
END_IF

// position trigger leaving station 0 for recovery
IF XTS.PositionTrigger[3].MoverPassedPosition THEN
	XTS.PositionTrigger[3].CurrentMover.SetVelocity(MainCommands.mediumVelocity).MoveToStation(XTS.Station[0]);
	XTS.PositionTrigger[3].MuteCurrent();
END_IF
END_ACTION

ACTION RecoverOneshot:

          // this action is called one time after the start command is issued
// it is intended to provide a single command to each mover to facilitate recovery
// other commands such as resetting counters and timers should also be carried out here

// clear any position trigers that were not consumed before the restart
XTS.System.MuteAllPositionTriggers();

// send all movers to station 0
XTS.System.CompleteMoverList.SetAllVelocity(MainCommands.mediumVelocity).MoveAllToStation( XTS.Station[0] );
//movers near station 0 (zone 0) need to first move away from the station
XTS.Zone[0].CurrentMoverList.MoveAllVelocity(MainCommands.lowVelocity);
// Restart statistics
XTS.System.ResetStatistics();

// Reinit nextStation
nextStation := 4;
END_ACTION

ACTION StationLogic:

          		(*Mover routing logic should be written here to define the system's operating behavior.
		Station implementations, Position Trigger logic, etc. In general, you can remove the example code
		here down to the short line break that looks like this: // ============= *)
	
        // Station 0 Logic
        IF XTS.Station[0].MoverInPosition THEN
            StationTimer[0](IN := TRUE, PT := T#1000MS);
            IF StationTimer[0].Q THEN
                XTS.Station[0].CurrentMover.MoveToStation(DestinationStation:= XTS.Station[1]);
            END_IF
        ELSE
            StationTimer[0](IN := FALSE);
        END_IF
		
        // Station 1 Logic		
        IF XTS.Station[1].MoverInPosition THEN
            StationTimer[1](IN := TRUE, PT := T#250MS);
            IF StationTimer[1].Q THEN
                XTS.Station[1].CurrentMover.MoveToStation(XTS.Station[nextStation]);
                nextStation := nextStation - 1;
                IF nextStation = 1 THEN
                    nextStation := 4;
                END_IF
            END_IF
        ELSE
            StationTimer[1](IN := FALSE);
        END_IF
		
		// Group of Stations 2, 3, and 4 Logic
        IF XTS.Station[2].MoverInPosition AND XTS.Station[3].MoverInPosition AND XTS.Station[4].MoverInPosition THEN
            StationTimer[2](IN := TRUE, PT := T#750MS);
            IF StationTimer[2].Q THEN
				StationTimer[2](IN := FALSE);
				
				XTS.Station[2].CurrentMover.MotionParameters:= XTS.InitialParameterSet;
				XTS.Station[3].CurrentMover.MotionParameters:= XTS.InitialParameterSet;
				XTS.Station[4].CurrentMover.MotionParameters:= XTS.InitialParameterSet;

                XTS.Station[2].CurrentMover.MoveVelocity(500);
                XTS.Station[3].CurrentMover.MoveVelocity(500);
                XTS.Station[4].CurrentMover.MoveVelocity(500);
				
            END_IF
        END_IF
		
        // Position Trigger 0 Logic
        IF XTS.PositionTrigger[0].MoverPassedPosition THEN
            XTS.PositionTrigger[0].CurrentMover.SetVelocity(MainCommands.lowVelocity);
			
			// To Call ApplicationMover addon Method/Properties/Variables, you must call Mover[] array index directly
			// Get MoverIndex for later use with ApplicationMover addons
			Trig0MoverIndex		:= XTS.PositionTrigger[0].CurrentMover.MoverIndex;
			
			// Call ApplicationMover Method/Properties/Variables using previously latched MoverIndex
			Trig0MoverPosLag	:= XTS.Mover[Trig0MoverIndex].PositionLag;
			
            XTS.PositionTrigger[0].MuteCurrent();
						
        END_IF
		
        // Position Trigger 1 Logic
        IF XTS.PositionTrigger[1].MoverPassedPosition THEN
			XTS.PositionTrigger[1].CurrentMover.SetAcceleration(5E2);
            XTS.PositionTrigger[1].CurrentMover.SetVelocity(MainCommands.highVelocity);
            XTS.PositionTrigger[1].MuteCurrent();
        END_IF

		// Position Trigger 2 Logic
        IF XTS.PositionTrigger[2].MoverPassedPosition THEN
			XTS.PositionTrigger[2].CurrentMover.SetAcceleration(1E4);
            XTS.PositionTrigger[2].CurrentMover.SetVelocity(MainCommands.lowVelocity);
            XTS.PositionTrigger[2].CurrentMover.MoveToStation(XTS.Station[0]);
            XTS.PositionTrigger[2].MuteCurrent();
        END_IF
END_ACTION

END_PROGRAM

// ---- POUs/ApplicationMover.TcPOU
// This function Block extends the Referenced Library Mover (FB), so the user can expand the capabilities of the XTS Mover Functions
FUNCTION_BLOCK ApplicationMover EXTENDS Mover
VAR_INPUT
END_VAR
VAR_OUTPUT
END_VAR
VAR
	_PositionLag: LREAL;
END_VAR

METHOD Cyclic : iMover
VAR_IN_OUT
	GroupReference	: AXES_GROUP_REF;
END_VAR
// Call Base Class (Mover) Cyclic Logic
SUPER^.Cyclic(GroupReference);

//======= 
// To Call ApplicationMover addon Method/Properties/Variables... 
//		you must call Mover[] array index directly, as Station/Zone/PositionTrig/SpeedTrig do not know about ApplicationMover add ons

// Add ApplicationMover specific code here

// example position lag property
_PositionLag:= THIS^.AxisReference.NcToPlc.PosDiff;

// Latch Errors

// Call Fbs Cyclically
END_METHOD

{attribute 'monitoring' := 'call'}
PROPERTY PositionLag : LREAL
GET
PositionLag:= _PositionLag;
END_GET
END_PROPERTY

END_FUNCTION_BLOCK

// ---- VISUs/Controls.TcVIS
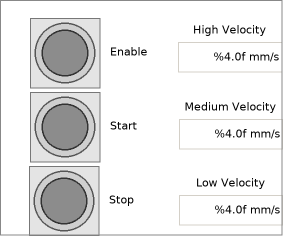
VISUALIZATION Controls  // 283x236
    PushSwitchLed (30,18 70x70), variable: MainCommands.Enable, behaviour: TOGGLE, style: Switch-PushSwitchLed-Gray
    Label (107,37 75x30), "Enable"
    Label (107,111 75x30), "Start"
    PushSwitchLed (30,92 70x70), variable: MainCommands.Start, behaviour: TOGGLE, style: Switch-PushSwitchLed-Gray
    Label (106,185 75x30), "Stop"
    PushSwitchLed (29,166 70x70), variable: MainCommands.Stop, behaviour: TOGGLE, style: Switch-PushSwitchLed-Gray
    Textfield (178,42 104x30), "%4.0f mm/s", text variable: MainCommands.highVelocity
        OnMouseClick: write the text variable via VisuDialogs.Numpad, min 1, max 2000, format %f.0
    Label (181,21 97x18), "High Velocity"
    Textfield (179,119 104x30), "%4.0f mm/s", text variable: MainCommands.mediumVelocity
        OnMouseClick: write the text variable via VisuDialogs.Numpad, min 1, max 2000, format %f.0
    Label (182,98 97x18), "Medium Velocity"
    Textfield (179,195 104x30), "%4.0f mm/s", text variable: MainCommands.lowVelocity
        OnMouseClick: write the text variable via VisuDialogs.Numpad, min 1, max 2000, format %f.0
    Label (182,174 97x18), "Low Velocity"
END_VISUALIZATION

// ---- VISUs/DiagnosticVisu.TcVIS
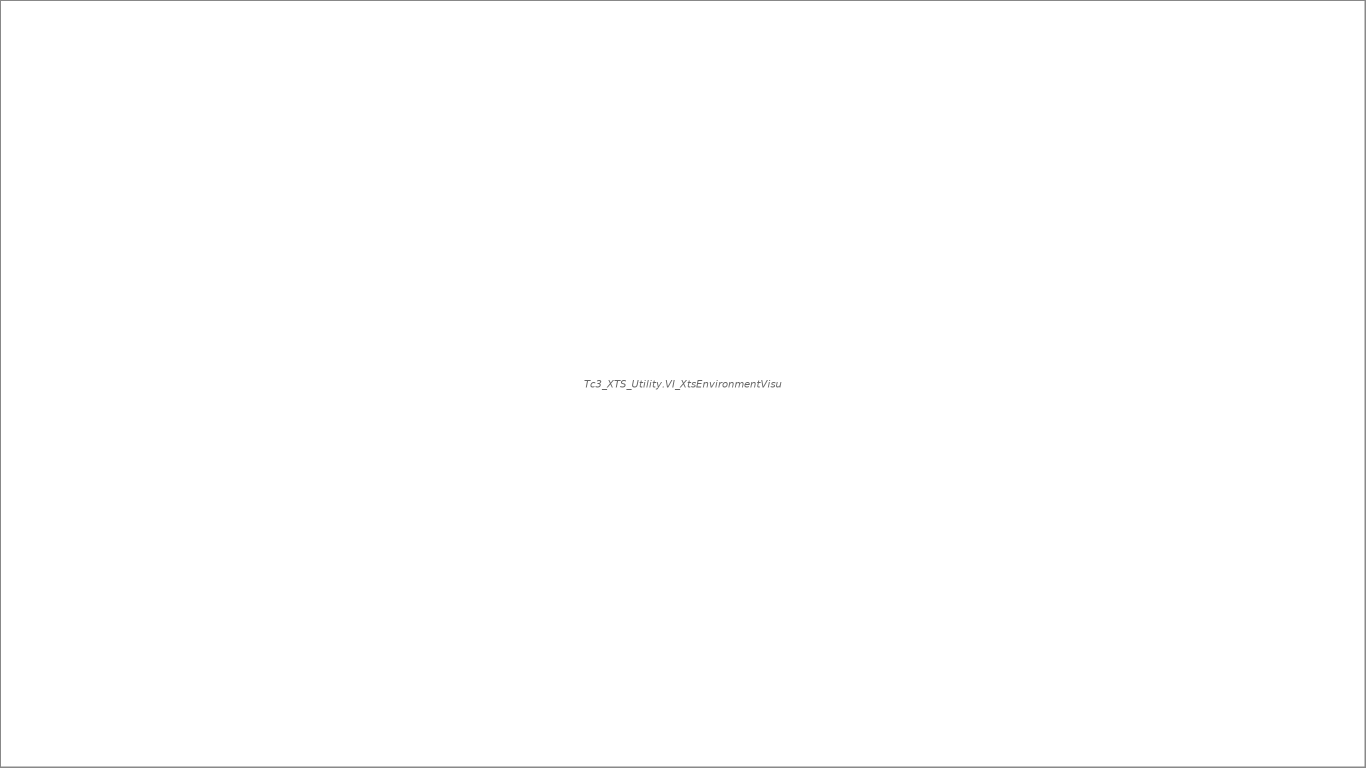
VISUALIZATION DiagnosticVisu  // 1366x768
    Frame (0,0 1366x768)
        shows Tc3_XTS_Utility.VI_XtsEnvironmentVisu()
END_VISUALIZATION
